FUNCTION_BLOCK Heating 
VAR_GENERIC CONSTANT
	ROOM_CAP		: UDINT := 20;
END_VAR

IMPLEMENTS I_Execute, I_Init
VAR_INPUT
	bPumpOverload	: BOOL;
	bBurnerOverload	: BOOL;

	rBoilerTemp		: LREAL := 60;
	rBoilerPressure	: LREAL := 1;
END_VAR
VAR_OUTPUT
	bPump			: BOOL;
	bBurner			: BOOL;
END_VAR
VAR
	_init			: Init(THIS^);
	_exe			: Execute(THIS^);
	_ctx			: Heating_Ctx;
	_tonPump		: TON;
	_tonBurner		: TON;	

	_entityStart	: EntityStart;
	_tag			: Tag := (Option := 'Heating');

	_smgr			: StateManager := (Proxy := _ctx.state.iMgr);
	
	_disabled		: Heating_State_Disabled(_ctx) := (Proxy := _ctx.state.iDisable);
	_safety         : Heating_State_Safety(_ctx) := (Proxy := _ctx.state.iSafety);
	_fault          : Heating_State_Fault(_ctx) := (Proxy := _ctx.state.iFault);
	_enabled        : Heating_State_Enabled(_ctx) := (Proxy := _ctx.state.iEnable);
	_pumping        : Heating_State_HeatingRoom(_ctx) := (Proxy := _ctx.state.iHeating);
	_heatup         : Heating_State_Heatup(_ctx) := (Proxy := _ctx.state.iHeatup);

	_enableEvent	: Signal := (Proxy := _ctx.priv.iOnEnable);
	_onRequestCall	: Heating_OnRequest(_ctx);
	_onRequest		: Receiver(_onRequestCall);
	
	_queue			: ArgQueue<ROOM_CAP> := (MutProxy := _ctx.priv.iQueue);
	
	_entityEnd		: EntityEnd;
END_VAR

METHOD Execute
// Inputs
_ctx.io.in.bBurnerOverload := bBurnerOverload;
_ctx.io.in.bPumpOverload := bPumpOverload;
_ctx.io.in.rBoilerPressure := rBoilerPressure;
_ctx.io.in.rBoilerTemp := rBoilerTemp;

// Outputs
_tonPump(IN := _ctx.io.out.bPump, PT := T#2S, Q => bPump);
_tonBurner(IN := _ctx.io.out.bBurner, PT := T#2S, Q => bBurner);

// SIMULATION

IF NOT sim.bTick THEN
	RETURN;
END_IF

// System temperature
IF bBurner THEN
	sim.rSystemTemperature := sim.rSystemTemperature + Sim.param.rSystemTemperatureRisePerBurner * Math.Random();
END_IF
sim.rSystemTemperature := sim.rSystemTemperature + Sim.param.rSystemTemperatureDropPassive * Math.Random();

IF sim.param.bToggleSystemTemperatureRise THEN
	sim.rSystemTemperature := sim.rSystemTemperature + Sim.param.rSystemTemperatureRise;
END_IF
IF sim.param.bToggleSystemTemperatureFall THEN
	sim.rSystemTemperature := sim.rSystemTemperature + Sim.param.rSystemTemperatureFall;
END_IF

IF sim.rSystemTemperature < 0 THEN
	sim.rSystemTemperature := 0;
ELSIF sim.rSystemTemperature > 100 THEN
	sim.rSystemTemperature := 100;
END_IF

sim.bFlow := bPump;

// System Pressure
IF sim.param.bToggleSystemPressureRise THEN
	sim.rSystemPressure := sim.rSystemPressure + Sim.param.rSystemPressureRise;
END_IF
IF sim.param.bToggleSystemPressureFall THEN
	sim.rSystemPressure := sim.rSystemPressure + Sim.param.rSystemPressureFall;
END_IF

IF sim.rSystemPressure < 0 THEN
	sim.rSystemPressure := 0;
ELSIF sim.rSystemPressure > 10 THEN
	sim.rSystemPressure := 10;
END_IF

// Write IO

rBoilerTemp := sim.rSystemTemperature;
rBoilerPressure := sim.rSystemPressure;
END_METHOD

METHOD Init
_smgr.Request(_disabled);
END_METHOD

END_FUNCTION_BLOCK

(* stored: Version 1.1.0.1
   POU Heating: Id {62f0b3a1-a792-4ec1-b14a-c56d60b72dc9}, SpecialFunc None
   Method Execute: Id {2db28cf4-24c2-48ef-813b-53c66671dd1a}
   Method Init: Id {cc8e1674-1a3f-478e-a1dc-45b6956a8d3e} *)
